// TIA Portal project "2022.04.24 电机正反转" (V17)

(* hardware
DEVICE "S7-1500/ET200MP station_1"  S7-1500 station
   slot 0: "导轨_0"  Rack  6ES7 590-1***0-0AA0
   slot 1: "PLC_1"  CPU 1516-3 PN/DP  6ES7 516-3AN00-0AB0  V1.7
      slot 3: "CPU 显示_1"  6ES7591-1BA00-0AA0
      slot 32768: "PROFINET 接口_1"  X1
         slot 32769: "端口_1"  X1 P1
         slot 32770: "端口_2"  X1 P2
      slot 33024: "PROFINET 接口_2"  X2
         slot 33025: "端口_1"  X2 P1
      slot 33280: "DP 接口_1"  X3
   slot 2: "DI 32x24VDC BA_1"  DI 32x24VDC BA  6ES7 521-1BL10-0AA0  V1.1
   slot 3: "DQ 32x24VDC/0.5A HF_1"  DQ 32x24VDC/0.5A HF  6ES7 522-1BL01-0AB0  V1.1
*)

// ===== PLC "PLC_1"  CPU 1516-3 PN/DP =====

VAR_GLOBAL   // PLC tag table "默认变量表"
   "正转按钮" AT %I0.0 : Bool;
   "反转按钮" AT %I0.1 : Bool;
   "停止按钮" AT %I0.2 : Bool;
   "按钮4" AT %I0.3 : Bool;
   "按钮5" AT %I0.4 : Bool;
   "按钮6" AT %I0.5 : Bool;
   "按钮7" AT %I0.6 : Bool;
   "按钮8" AT %I0.7 : Bool;
   "按钮9" AT %I1.0 : Bool;
   "按钮10" AT %I1.1 : Bool;
   "按钮11" AT %I1.2 : Bool;
   "电机正转" AT %Q0.0 : Bool;
   "电机反转" AT %Q0.1 : Bool;
   "指示灯3" AT %Q0.2 : Bool;
   "指示灯4" AT %Q0.3 : Bool;
   "指示灯5" AT %Q0.4 : Bool;
   "指示灯6" AT %Q0.5 : Bool;
   "指示灯7" AT %Q0.6 : Bool;
   "指示灯8" AT %Q0.7 : Bool;
   "指示灯9" AT %Q1.0 : Bool;
   "指示灯10" AT %Q1.1 : Bool;
   "指示灯11" AT %Q1.2 : Bool;
   "指示灯12" AT %Q1.3 : Bool;
   "Tag_1" AT %M0.0 : Bool;
END_VAR

FUNCTION "电机控制LAD" : Void   // FC1, LAD
{ S7_Optimized_Access := 'TRUE' }
VERSION : 0.1
BEGIN

REGION Network 1: 正转按钮
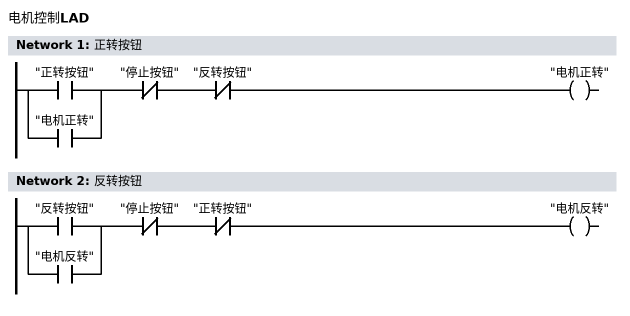
   RUNG wire#powerrail
      Contact( "正转按钮" )
      wire#w1
      I_Contact( "停止按钮" )
      I_Contact( "反转按钮" )
      Coil( "电机正转" )
   END_RUNG
   RUNG wire#powerrail
      Contact( "电机正转" )
   END_RUNG wire#w1
   // the same network as SCL:
   "电机正转" := ("正转按钮" OR "电机正转") AND NOT "停止按钮" AND NOT "反转按钮";
END_REGION

REGION Network 2: 反转按钮
   RUNG wire#powerrail
      Contact( "反转按钮" )
      wire#w1
      I_Contact( "停止按钮" )
      I_Contact( "正转按钮" )
      Coil( "电机反转" )
   END_RUNG
   RUNG wire#powerrail
      Contact( "电机反转" )
   END_RUNG wire#w1
   // the same network as SCL:
   "电机反转" := ("反转按钮" OR "电机反转") AND NOT "停止按钮" AND NOT "正转按钮";
END_REGION
END_FUNCTION

FUNCTION "电机控制-FBD" : Void   // FC2, FBD
{ S7_Optimized_Access := 'TRUE' }
VERSION : 0.1
BEGIN

REGION Network 1
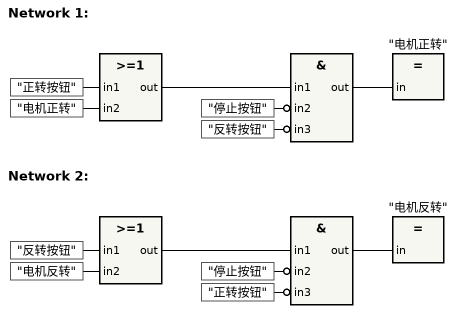
   "电机正转" := ("正转按钮" OR "电机正转") AND NOT "停止按钮" AND NOT "反转按钮";
END_REGION

REGION Network 2
   "电机反转" := ("反转按钮" OR "电机反转") AND NOT "停止按钮" AND NOT "正转按钮";
END_REGION
END_FUNCTION

FUNCTION "电机控制SCL" : Void   // FC3, SCL
{ S7_Optimized_Access := 'TRUE' }
VERSION : 0.1
BEGIN
   //正转控制

   IF "正转按钮" THEN
       "电机正转" :=1
       ;
   END_IF;
   IF "停止按钮" = TRUE OR "反转按钮" = TRUE THEN
       "电机正转" := 0
       ;
   END_IF;

   //反转控制
   IF "反转按钮" THEN
       "电机反转" := 1
       ;
   END_IF;
   IF "停止按钮" = TRUE OR "正转按钮" = TRUE THEN
       "电机反转" := 0
       ;
   END_IF;
END_FUNCTION

ORGANIZATION_BLOCK "Main"   // OB1, LAD, ProgramCycle
TITLE = "Main Program Sweep (Cycle)"
{ S7_Optimized_Access := 'TRUE' }
VERSION : 0.1
   VAR_INPUT
      Initial_Call : Bool;   // Initial call of this OB
      Remanence : Bool;   // =True, if remanent data are available
   END_VAR
   VAR_TEMP
      "123" : Byte;
   END_VAR
BEGIN

REGION Network 1
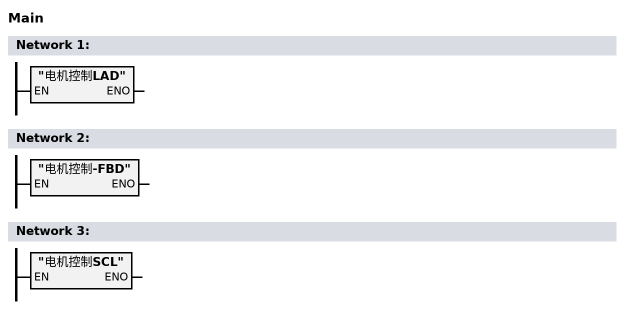
   RUNG wire#powerrail
      "电机控制LAD"()
   END_RUNG
   // the same network as SCL:
   "电机控制LAD"();
END_REGION

REGION Network 2
   RUNG wire#powerrail
      "电机控制-FBD"()
   END_RUNG
   // the same network as SCL:
   "电机控制-FBD"();
END_REGION

REGION Network 3
   RUNG wire#powerrail
      "电机控制SCL"()
   END_RUNG
   // the same network as SCL:
   "电机控制SCL"();
END_REGION
END_ORGANIZATION_BLOCK